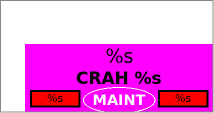
VISUALIZATION AminCRAH  // 214x113
VAR_INPUT
	idCrah : WSTRING;
	Offline : BOOL;
	Alarm : BOOL;
	Enable: BOOL;
	Running: BOOL;
	Inhibited : BOOL;
	Maintenance : BOOL;		
	HOA : WORD;
	Isolator1 : BOOL;
	Isolator2 : BOOL;
	DeactivateIso2 : BOOL;
END_VAR
    Rectangle (24,43 190x70), colour toggle: Enable
    Rectangle (24,43 190x70), colour toggle: Enable, invisible if: Not Running
    Rectangle (24,43 190x70), colour toggle: Enable, invisible if: Not Inhibited
    Rectangle (24,43 190x70), colour toggle: Enable, invisible if: Not Offline
    Rectangle (24,43 190x70), "CRAH %s", text variable: idCrah, colour toggle: Enable, invisible if: Not Inhibited
    Rectangle (84,46 71x21), "%s", text list: 'CRAH_Status', text index: HOA
    Ellipse (83,87 72x26), "MAINT", invisible if: Not Inhibited
    Rectangle (30,90 50x17), "%s", colour toggle: Isolator1, text list: 'CRAH_Isolator_Status', text index: Isolator1
    Rectangle (158,90 50x17), "%s", colour toggle: Isolator2, text list: 'CRAH_Isolator_Status', text index: Isolator2
END_VISUALIZATION

(* stored: Version 1.1.0.1, ProductVersion 3.1.4024.12
   Visu AminCRAH: Id {354e3d56-b88a-4f66-957c-c93b263eb97b} *)
